// TwinCAT 3 PLC project PLC
// ProgramVersion: 3.1.4026.23
// libraries:
//   Tc2_EtherCAT, * (Beckhoff Automation GmbH)
//   Tc2_Standard, * (Beckhoff Automation GmbH)
//   Tc2_System, * (Beckhoff Automation GmbH)
//   Tc3_RealtimeMonitoring, * (Beckhoff Automation GmbH)
// project tree:
//   DUTs/ F_ConsumeTime.TcPOU
//   / PlcTask.TcTTO
//   POUs/ MAIN.TcPOU
// real-time tasks:
//   TASK PlcTask: cycle T#1ms, priority 20, ADS port 350

CONFIGURATION PLC
    RESOURCE PLC ON TwinCAT3
        TASK PlcTask(INTERVAL := T#1ms, PRIORITY := 20);
        PROGRAM MAIN WITH PlcTask : MAIN;
    END_RESOURCE
END_CONFIGURATION

// ---- POUs/MAIN.TcPOU
PROGRAM MAIN
VAR
	Execute : BOOL;
	Step	: UDINT;
	LogMark : FB_RTMon_LogMark;
END_VAR
(*
In Realtime monitor,
Add a user contex:
Context ID : 851 (0x353)

Add new user group :
Group ID: 0

*)

IF Execute THEN
	Execute := FALSE;
	LogMark.LogStart(0, 0);
	LogMark.LogTrigger(0, 0);
	F_ConsumeTime(100);
	LogMark.LogMark(0, 10);
	F_ConsumeTime(100);
	LogMark.LogMark(0, 20);
	F_ConsumeTime(100);
	LogMark.LogStop(0, 0);
END_IF

END_PROGRAM

// ---- DUTs/F_ConsumeTime.TcPOU
FUNCTION F_ConsumeTime
VAR_INPUT
	Us		:UDINT;
END_VAR
VAR
		tCurr, tEnd : T_DCTIME64;
END_VAR

tCurr := F_GetActualDcTime64();
tEnd  := tCurr + (Us * EC_DCTIME_TICKSPERMSEC64 / 1000);
WHILE (tCurr < tEnd) DO
	tCurr := F_GetActualDcTime64();
END_WHILE

END_FUNCTION
